{attribute 'qualified_only'}
{attribute 'strict'}
{attribute 'to_string'}
TYPE E_AirState :
(
	UNKNOWN := 0,
	DIRTY,
	CLEAN
);
END_TYPE

(* stored: Version 1.1.0.1, ProductVersion 3.1.4024.12
   DUT E_AirState: Id {4bb3c501-2666-4d89-b793-16d979d0712b} *)
